TEXTLIST TL_Aktoren
  0 = 'keine Aktion'
  1 = 'Aktor1 Vor'
  2 = 'Aktor1 Zurück'
  3 = 'Aktor2 Vor'
  4 = 'Aktor2 Zurück'
  5 = 'Aktor3 Vor'
  6 = 'Aktor3 Zurück'
  7 = 'Aktor4 Vor'
  8 = 'Aktor4 Zurück'
  9 = 'Aktor5 Vor'
  10 = 'Aktor5 Zurück'
  11 = 'Aktor6 Vor'
  12 = 'Aktor6 Zurück'
  13 = 'teilAnwesend'
  14 = 'Ext. Gerät bereit'
  15 = 'Ext. Gerät starten'
  16 = 'warten'
   = ''
END_TEXTLIST

(* stored: Version 1.1.0.1, ProductVersion 3.1.4024.12
   TextList TL_Aktoren: Id {7c530262-d051-4597-8330-6f0d637c777a} *)
